(* CODESYS project intersection.project
   Title: mehatronika
   Version: 0.0.0.0
   Author: jasar

Project tree, tasks and I/O mapping:
  XBTGT7340 : XBTGT7340, Schneider Electric, order no. XBTGT7340, version 3.5.3.54
    HMI Application
    COM2
      SoMachine_Network_Manager4 : SoMachine-Network Manager, Schneider Electric, version 4.0.0.2
    USB
      SoMachine_Network_Manager6 : SoMachine-Network Manager, Schneider Electric, version 4.0.0.2
    COM1
      SoMachine_Network_Manager3 : SoMachine-Network Manager, Schneider Electric, version 4.0.0.2
    Ethernet
      SoMachine_Network_Manager5 : SoMachine-Network Manager, Schneider Electric, version 4.0.0.2
  MyController : TM241CE24T/U, Schneider Electric, order no. TM241CE24T/U, version 4.0.6.18
    application Application
      task MAST (cyclic, interval 20 ms, priority 15, watchdog 100 ms x 1) calls POU
      task Task (cyclic, interval t#500ms, priority 1) calls POU_1
      global variables GVL
      program POU [SFC]: Init_entry, Init_active, Step0_entry, Step0_active, Stage_3_entry, Stage_3_active, Stage_4_entry, Stage_4_active, Stage_5_entry, Stage_5_active, Stage_6_entry, Stage_6_active, Stage_7_entry, Stage_7_active, Stage_8_entry, Stage_8_active, Stage_9_entry, Stage_9_active, Stage_10_entry, Stage_10_active, Stage_11_entry, Stage_11_active, Stage_12_entry, Stage_12_active, Stage_13_entry, Stage_13_active, Stage_14_entry, Stage_14_active, Stage_15_entry, Stage_15_active, Stage_16_entry, Stage_16_active, Stage_17_entry, Stage_17_active, Stage_18_entry, Stage_18_active, Stage_19_entry, Stage_19_active, Stage_20_entry, Stage_20_active, Stage_21_entry, Stage_21_active, Stage_22_entry, Stage_22_active, Stage_23_entry, Stage_23_active, Stage_24_entry, Stage_24_active
      program POU_1 [ST]
      Symbols
    DI : Digital Inputs, Schneider Electric, version 4.0.6.18
        input  iwDI_IW0 : WORD  // IW0
        input  ibDI_IB1 : BYTE  // IB1
    DQ : Digital Outputs, Schneider Electric, version 4.0.6.18
        output qwDQ_QW0 : WORD  // QW0
        output qbDQ_QB1 : BYTE  // QB1
    Counters : Counters, Schneider Electric, version 4.0.6.18
    Pulse_Generators : Pulse Generators, Schneider Electric, version 4.0.6.18
    Cartridge_1 : Cartridge, Schneider Electric, version 4.0.6.18
    IO_Bus : IO bus - TM3, Schneider Electric, version 4.0.6.18
    COM_Bus : COM bus, Schneider Electric, version 4.0.6.18
    Ethernet_1 : Ethernet Network, Schneider Electric, version 4.0.6.18
    Serial_Line_1 : Serial line, Schneider Electric, version 4.0.6.18
      SoMachine_Network_Manager : SoMachine-Network Manager, Schneider Electric, version 4.0.0.2
    Serial_Line_2 : Serial line, Schneider Electric, version 4.0.6.18
      Modbus_Manager : Modbus Manager, Schneider Electric, version 4.0.0.2
  Vijeo Designer Project Container Data
  Vijeo Designer Project Container
*)

// MyController/Application/GVL
VAR_GLOBAL
END_VAR
VAR_GLOBAL
	pomoc: BOOL;
	blinker: BOOL;
	tajmer: TOF;
	okidac: BOOL;
	pjesak8: BOOL := TRUE;
	pjesak7: BOOL := TRUE;
	pjesak6: BOOL := FALSE;
	pjesak5: BOOL := FALSE;
	pjesak4: BOOL := TRUE;
	pjesak3: BOOL := TRUE;
	pjesak2: BOOL := FALSE;
	pjesak1: BOOL := FALSE;
	semafor8_zelena: BOOL;
	semafor8_zuta: BOOL;
	semafor8_crvena: BOOL := TRUE;
	semafor7_zelena: BOOL;
	semafor7_zuta: BOOL;
	semafor7_crvena: BOOL := TRUE;
	semafor6_zelena: BOOL;
	semafor6_zuta: BOOL;
	semafor6_crvena: BOOL;
	semafor5_zelena: BOOL;
	semafor5_zuta: BOOL;
	semafor5_crvena: BOOL := TRUE;
	semafor4_zelena: BOOL;
	semafor4_zuta: BOOL;
	semafor4_crvena: BOOL := TRUE;
	semafor3_zelena: BOOL;
	semafor3_zuta: BOOL;
	semafor3_crvena: BOOL := TRUE;
	semafor2_zelena: BOOL;
	semafor2_zuta: BOOL;
	semafor2_crvena: BOOL;
	semafor1_zelena: BOOL;
	semafor1_zuta: BOOL;
	semafor1_crvena: BOOL := TRUE;
END_VAR

// MyController/Application/POU
PROGRAM POU
VAR
	semfor8_zuta: BOOL;
END_VAR

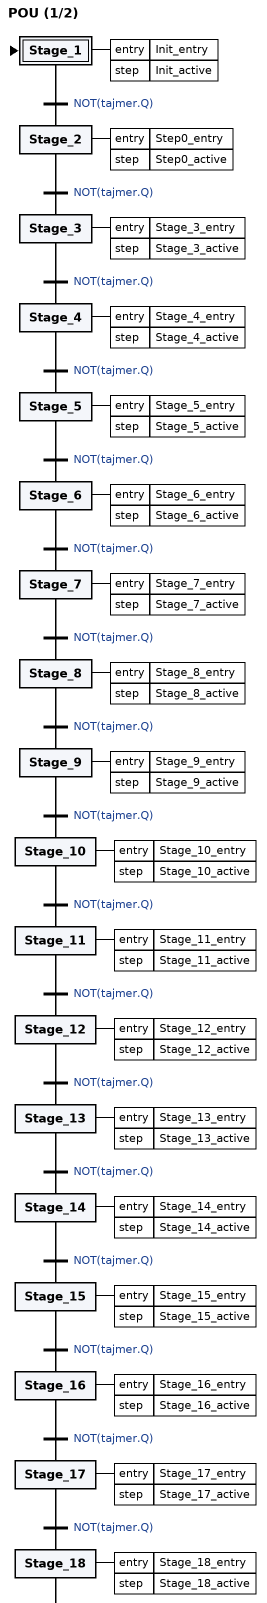
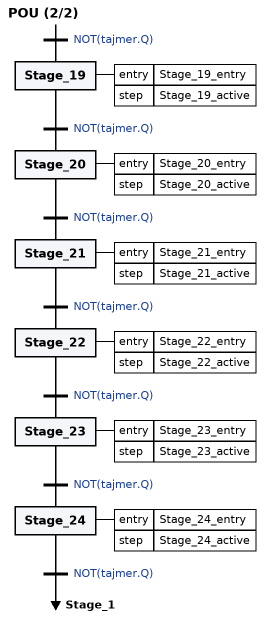
INITIAL_STEP Stage_1:
    Init_entry(P1);  // entry action
    Init_active(N);  // step action
END_STEP
TRANSITION FROM Stage_1 TO Stage_2
    := NOT(tajmer.Q);
END_TRANSITION
STEP Stage_2:
    Step0_entry(P1);  // entry action
    Step0_active(N);  // step action
END_STEP
TRANSITION FROM Stage_2 TO Stage_3
    := NOT(tajmer.Q);
END_TRANSITION
STEP Stage_3:
    Stage_3_entry(P1);  // entry action
    Stage_3_active(N);  // step action
END_STEP
TRANSITION FROM Stage_3 TO Stage_4
    := NOT(tajmer.Q);
END_TRANSITION
STEP Stage_4:
    Stage_4_entry(P1);  // entry action
    Stage_4_active(N);  // step action
END_STEP
TRANSITION FROM Stage_4 TO Stage_5
    := NOT(tajmer.Q);
END_TRANSITION
STEP Stage_5:
    Stage_5_entry(P1);  // entry action
    Stage_5_active(N);  // step action
END_STEP
TRANSITION FROM Stage_5 TO Stage_6
    := NOT(tajmer.Q);
END_TRANSITION
STEP Stage_6:
    Stage_6_entry(P1);  // entry action
    Stage_6_active(N);  // step action
END_STEP
TRANSITION FROM Stage_6 TO Stage_7
    := NOT(tajmer.Q);
END_TRANSITION
STEP Stage_7:
    Stage_7_entry(P1);  // entry action
    Stage_7_active(N);  // step action
END_STEP
TRANSITION FROM Stage_7 TO Stage_8
    := NOT(tajmer.Q);
END_TRANSITION
STEP Stage_8:
    Stage_8_entry(P1);  // entry action
    Stage_8_active(N);  // step action
END_STEP
TRANSITION FROM Stage_8 TO Stage_9
    := NOT(tajmer.Q);
END_TRANSITION
STEP Stage_9:
    Stage_9_entry(P1);  // entry action
    Stage_9_active(N);  // step action
END_STEP
TRANSITION FROM Stage_9 TO Stage_10
    := NOT(tajmer.Q);
END_TRANSITION
STEP Stage_10:
    Stage_10_entry(P1);  // entry action
    Stage_10_active(N);  // step action
END_STEP
TRANSITION FROM Stage_10 TO Stage_11
    := NOT(tajmer.Q);
END_TRANSITION
STEP Stage_11:
    Stage_11_entry(P1);  // entry action
    Stage_11_active(N);  // step action
END_STEP
TRANSITION FROM Stage_11 TO Stage_12
    := NOT(tajmer.Q);
END_TRANSITION
STEP Stage_12:
    Stage_12_entry(P1);  // entry action
    Stage_12_active(N);  // step action
END_STEP
TRANSITION FROM Stage_12 TO Stage_13
    := NOT(tajmer.Q);
END_TRANSITION
STEP Stage_13:
    Stage_13_entry(P1);  // entry action
    Stage_13_active(N);  // step action
END_STEP
TRANSITION FROM Stage_13 TO Stage_14
    := NOT(tajmer.Q);
END_TRANSITION
STEP Stage_14:
    Stage_14_entry(P1);  // entry action
    Stage_14_active(N);  // step action
END_STEP
TRANSITION FROM Stage_14 TO Stage_15
    := NOT(tajmer.Q);
END_TRANSITION
STEP Stage_15:
    Stage_15_entry(P1);  // entry action
    Stage_15_active(N);  // step action
END_STEP
TRANSITION FROM Stage_15 TO Stage_16
    := NOT(tajmer.Q);
END_TRANSITION
STEP Stage_16:
    Stage_16_entry(P1);  // entry action
    Stage_16_active(N);  // step action
END_STEP
TRANSITION FROM Stage_16 TO Stage_17
    := NOT(tajmer.Q);
END_TRANSITION
STEP Stage_17:
    Stage_17_entry(P1);  // entry action
    Stage_17_active(N);  // step action
END_STEP
TRANSITION FROM Stage_17 TO Stage_18
    := NOT(tajmer.Q);
END_TRANSITION
STEP Stage_18:
    Stage_18_entry(P1);  // entry action
    Stage_18_active(N);  // step action
END_STEP
TRANSITION FROM Stage_18 TO Stage_19
    := NOT(tajmer.Q);
END_TRANSITION
STEP Stage_19:
    Stage_19_entry(P1);  // entry action
    Stage_19_active(N);  // step action
END_STEP
TRANSITION FROM Stage_19 TO Stage_20
    := NOT(tajmer.Q);
END_TRANSITION
STEP Stage_20:
    Stage_20_entry(P1);  // entry action
    Stage_20_active(N);  // step action
END_STEP
TRANSITION FROM Stage_20 TO Stage_21
    := NOT(tajmer.Q);
END_TRANSITION
STEP Stage_21:
    Stage_21_entry(P1);  // entry action
    Stage_21_active(N);  // step action
END_STEP
TRANSITION FROM Stage_21 TO Stage_22
    := NOT(tajmer.Q);
END_TRANSITION
STEP Stage_22:
    Stage_22_entry(P1);  // entry action
    Stage_22_active(N);  // step action
END_STEP
TRANSITION FROM Stage_22 TO Stage_23
    := NOT(tajmer.Q);
END_TRANSITION
STEP Stage_23:
    Stage_23_entry(P1);  // entry action
    Stage_23_active(N);  // step action
END_STEP
TRANSITION FROM Stage_23 TO Stage_24
    := NOT(tajmer.Q);
END_TRANSITION
STEP Stage_24:
    Stage_24_entry(P1);  // entry action
    Stage_24_active(N);  // step action
END_STEP
TRANSITION FROM Stage_24 TO Stage_1
    := NOT(tajmer.Q);
END_TRANSITION

ACTION Init_entry:
semafor6_zuta := FALSE;
semafor6_crvena := FALSE;
semafor6_zelena := TRUE;
semafor2_zelena := TRUE;
okidac := TRUE;
END_ACTION

ACTION Init_active:
tajmer(IN:= okidac, PT := T#73S);
okidac := FALSE;
END_ACTION

ACTION Step0_entry:
blinker := FALSE;
okidac := TRUE;
END_ACTION

ACTION Step0_active:
tajmer (IN := okidac, PT := T#3S);
okidac := FALSE;
semafor2_zelena := blinker;
END_ACTION

ACTION Stage_3_entry:
semafor2_zelena := FALSE;
semafor2_zuta := TRUE;
okidac := TRUE;
END_ACTION

ACTION Stage_3_active:
tajmer(IN := okidac, PT := T#2S);
okidac := FALSE;
END_ACTION

ACTION Stage_4_entry:
semafor2_zuta := FALSE;
semafor2_crvena := TRUE;
semafor5_zuta := TRUE;
semafor5_crvena := TRUE;

pjesak2 := TRUE;
pjesak6 := TRUE;

okidac := TRUE;
END_ACTION

ACTION Stage_4_active:
tajmer(IN := okidac, PT := T#1S);
okidac := FALSE;
END_ACTION

ACTION Stage_5_entry:
semafor5_zelena := TRUE;
semafor5_zuta := FALSE;
semafor5_crvena := FALSE;

okidac := TRUE;
END_ACTION

ACTION Stage_5_active:
tajmer(IN := okidac, PT := T#6S);
okidac := FALSE;
END_ACTION

ACTION Stage_6_entry:
blinker := FALSE;
okidac := TRUE;
END_ACTION

ACTION Stage_6_active:
tajmer(IN := okidac, PT := T#3S);
okidac := FALSE;
semafor6_zelena := blinker;
semafor5_zelena := blinker;
END_ACTION

ACTION Stage_7_entry:
semafor6_zelena := FALSE;
semafor6_zuta := TRUE;

semafor5_zelena := FALSE;
semafor5_zuta := TRUE;

pjesak3 := FALSE;
pjesak7 := FALSE;

okidac := TRUE;
END_ACTION

ACTION Stage_7_active:
tajmer(IN := okidac, PT := T#2S);
okidac := FALSE;
END_ACTION

ACTION Stage_8_entry:
semafor6_zuta := FALSE;
semafor6_crvena := TRUE;

semafor5_zuta := FALSE;
semafor5_crvena := TRUE;

pjesak4 := TRUE;
pjesak8 := TRUE;

semafor4_crvena := TRUE;
semafor3_crvena := TRUE;
semafor4_zuta := TRUE;
semafor3_zuta := TRUE;

okidac := TRUE;
END_ACTION

ACTION Stage_8_active:
tajmer(IN := okidac, PT := T#1S);

okidac := FALSE;
END_ACTION

ACTION Stage_9_entry:
semafor4_crvena := FALSE;
semafor3_crvena := FALSE;
semafor4_zuta := FALSE;
semafor3_zuta := FALSE;

semafor4_zelena := TRUE;
semafor3_zelena := TRUE;

pjesak1 := TRUE;
pjesak5 := TRUE;


okidac := TRUE;
END_ACTION

ACTION Stage_9_active:
tajmer(IN := okidac, PT := T#6S);
okidac := FALSE;
END_ACTION

ACTION Stage_10_entry:
blinker := FALSE;

okidac := TRUE;
END_ACTION

ACTION Stage_10_active:
tajmer(IN := okidac, PT := T#3S);

okidac := FALSE;
semafor3_zelena := blinker;
END_ACTION

ACTION Stage_11_entry:
semafor3_zelena := FALSE;
semafor3_zuta := TRUE;

pjesak8 := FALSE;
pjesak4 := FALSE;

okidac := TRUE;
END_ACTION

ACTION Stage_11_active:
tajmer(IN := okidac, PT := T#2S);

okidac := FALSE;
END_ACTION

ACTION Stage_12_entry:
semafor3_zuta := FALSE;
semafor3_crvena := TRUE;

semafor8_crvena := TRUE;
semafor8_zuta := TRUE;

okidac := TRUE;
END_ACTION

ACTION Stage_12_active:
tajmer(IN := okidac, PT := T#1S);

okidac := FALSE;
END_ACTION

ACTION Stage_13_entry:
semafor8_crvena := FALSE;
semafor8_zuta := FALSE;
semafor8_zelena := TRUE;

okidac := TRUE;
END_ACTION

ACTION Stage_13_active:
tajmer(IN := okidac, PT := T#13S);

okidac := FALSE;
END_ACTION

ACTION Stage_14_entry:
blinker := FALSE;

okidac := TRUE;
END_ACTION

ACTION Stage_14_active:
tajmer(IN := okidac, PT := T#3S);

okidac := FALSE;
semafor4_zelena := blinker;
END_ACTION

ACTION Stage_15_entry:
semafor4_zelena := FALSE;
semafor4_zuta := TRUE;

okidac := TRUE;
END_ACTION

ACTION Stage_15_active:
tajmer(IN := okidac, PT := T#2S);

okidac := FALSE;
END_ACTION

ACTION Stage_16_entry:
semafor4_zuta := FALSE;
semafor4_crvena := TRUE;
semafor7_crvena := TRUE;
semafor7_zuta := TRUE;

pjesak3 := TRUE;
pjesak7 := TRUE;

okidac := TRUE;
END_ACTION

ACTION Stage_16_active:
tajmer(IN := okidac, PT := T#1S);

okidac := FALSE;
END_ACTION

ACTION Stage_17_entry:
semafor7_crvena := FALSE;
semafor7_zuta := FALSE;
semafor7_zelena := TRUE;

okidac := TRUE;
END_ACTION

ACTION Stage_17_active:
tajmer(IN := okidac, PT := T#6S);

okidac := FALSE;
END_ACTION

ACTION Stage_18_entry:
blinker := FALSE;
okidac := TRUE;
END_ACTION

ACTION Stage_18_active:
tajmer(IN := okidac, PT := T#3S);

okidac := FALSE;

semafor7_zelena := blinker;
semafor8_zelena := blinker;
END_ACTION

ACTION Stage_19_entry:
semafor7_zelena := FALSE;
semafor8_zelena := FALSE;

semafor7_zuta := TRUE;
semafor8_zuta := TRUE;

pjesak6 := FALSE;
pjesak2 := FALSE;

okidac := TRUE;
END_ACTION

ACTION Stage_19_active:
tajmer(IN := okidac, PT := T#2S);

okidac := FALSE;
END_ACTION

ACTION Stage_20_entry:
semafor7_zuta := FALSE;
semafor8_zuta := FALSE;

semafor7_crvena := TRUE;
semafor8_crvena := TRUE;

semafor2_zuta := TRUE;
semafor1_zuta := TRUE;

pjesak4 := TRUE;
pjesak8 := TRUE;

okidac := TRUE;
END_ACTION

ACTION Stage_20_active:
tajmer(IN := okidac, PT := T#1S);

okidac := FALSE;
END_ACTION

ACTION Stage_21_entry:
semafor2_zuta := FALSE;
semafor1_zuta := FALSE;

semafor2_crvena := FALSE;
semafor1_crvena := FALSE;

semafor2_zelena := TRUE;
semafor1_zelena := TRUE;

okidac := TRUE;
END_ACTION

ACTION Stage_21_active:
tajmer(IN := okidac, PT := T#6S);

okidac := FALSE;
END_ACTION

ACTION Stage_22_entry:
blinker := FALSE;

okidac := TRUE;
END_ACTION

ACTION Stage_22_active:
tajmer(IN := okidac, PT := T#3S);

semafor1_zelena := blinker;

okidac := FALSE;
END_ACTION

ACTION Stage_23_entry:
semafor1_zelena := FALSE;
semafor1_zuta := TRUE;

pjesak5 := FALSE;
pjesak1 := FALSE;

okidac := TRUE;
END_ACTION

ACTION Stage_23_active:
tajmer(IN := okidac, PT := T#2S);

okidac := FALSE;
END_ACTION

ACTION Stage_24_entry:
semafor1_zuta := FALSE;
semafor1_crvena := TRUE;

semafor6_zuta := TRUE;

okidac := TRUE;
END_ACTION

ACTION Stage_24_active:
tajmer(IN := okidac, PT := T#1S);

okidac := FALSE;
END_ACTION

END_PROGRAM

// MyController/Application/POU_1
PROGRAM POU_1
VAR
END_VAR

blinker := NOT(BLINKER);

END_PROGRAM
